{attribute 'GeneratedUsingTerminal: EK1322-0000-0017'}
{attribute addProperty BoxType "EK1322-0000-0017"}
{attribute addProperty Id "Status_UsAT %I*Status_Us_B1E819A21Status_UpAT %I*Status_Up_B1E819A21WcStateAT %I*WcState_9091E0EB2InfoDataAT %I*InfoData_6F19DB2B2"}
{attribute addProperty CRC "1807752468"}
{attribute addProperty Size "6"}
TYPE EK1322_6BC01D14 EXTENDS EtcSlaveTerminalBase_947E5A46 :
STRUCT
	{attribute addProperty Name "Status_Us"}
	Status_Us : Status_Us_B1E819A2;
	{attribute addProperty Name "Status_Up"}
	Status_Up : Status_Up_B1E819A2;
	{attribute addProperty Name "WcState"}
	WcState : WcState_9091E0EB;
	{attribute addProperty Name "InfoData"}
	InfoData : InfoData_6F19DB2B;
END_STRUCT
END_TYPE

(* stored: Version 1.2.0.0, ProductVersion 3.1.4024.9
   DUT EK1322_6BC01D14: Id {de22f9ff-c9c2-4f5d-b20b-8a78b3baa6a4} *)
